PROGRAM SlowPRG_1
VAR
	bolPlcStartupDone: BOOL := FALSE;
	bolHostInitDone : BOOL := FALSE;
	bolInitDone : BOOL := FALSE;
	jj:INT;
	bolCtrlRst: BOOL;
	
	fbAlm_Man: FB_Alm_Man; // alarm manager
END_VAR

(*__________________________________________________________________________________________________
¦	
¦	Vistaprint Schweiz GmbH
¦	CH - 8401 Winterthur
¦
¦	www.vistaprint.ch - info@vistaprint.ch
¦___________________________________________________________________________________________________

Function desription:
call of all controller (FUB) for the slow task class.


History:
Version		Date			Author		Comment
---------------------------------------------------------------------------------------------------
0.00.1		24.05.2013		AVME/KVO	Start history
0.00.2		07.11.2013		AVME/KVO	Add local variabel fbAlm_Man, Add set all initialized controller FB the property of the alarm manager adress 
0.00.3		08.11.2013		AVME/KVO	global g_p_fbAlm_Man adress assigned
___________________________________________________________________________________________________*)


// -----------------------------------------------------------------------------------------------
// Initialize the PLC Parameter and check the PLC health
// -----------------------------------------------------------------------------------------------
IF (NOT bolPlcStartupDone) THEN

	// set all initialized controller FB the property of the alarm manager adress 
	Base_PLC.setAllCtrlAlarmFB(pCtrlInst := ADR(g_a_pCtrlInst[0]), pAlarmCtrl := ADR(fbAlm_Man), uinCtrlInstLength := INT_TO_UINT(E_CtrlId.E_CtrlIdMax));
	g_p_fbAlm_Man := ADR(fbAlm_Man);
	bolPlcStartupDone := TRUE;	
END_IF
// -----------------------------------------------------------------------------------------------


// -----------------------------------------------------------------------------------------------
// The host system is downloading all parameter at startup. 
// bolPlcStartupDone will be set to true after the Host is done with the initialization
// -----------------------------------------------------------------------------------------------
IF (bolPlcStartupDone AND (NOT bolHostInitDone) AND NOT bolInitDone) THEN
	bolHostInitDone := TRUE;
END_IF
// -----------------------------------------------------------------------------------------------


// -----------------------------------------------------------------------------------------------
// Start PLC code initialization
// -----------------------------------------------------------------------------------------------
IF NOT bolInitDone AND bolPlcStartupDone AND bolHostInitDone THEN
	
	// init	
	bolInitDone := TRUE;
END_IF
// -----------------------------------------------------------------------------------------------

// -----------------------------------------------------------------------------------------------
// Normal Run mode after all the initialization is done
// -----------------------------------------------------------------------------------------------
IF (bolInitDone AND bolPlcStartupDone AND bolHostInitDone) THEN
	
	//****************************************************************************************************
	// cyclic controller calls
	//****************************************************************************************************
	// call alarm message handler
	fbAlm_Man(bolCtrlRst:= bolCtrlRst);
	IF (bolCtrlRst) THEN
		FOR jj:=0 TO E_CtrlId.E_CtrlIdMax BY 1 DO
			IF (g_a_pCtrlCIf[jj]<>0) THEN // check if entry exist
				g_a_pCtrlCIf[jj]^.Job.bolAlmReset := TRUE;
			END_IF
		END_FOR
		bolCtrlRst := FALSE;
	END_IF

END_IF
// -----------------------------------------------------------------------------------------------

END_PROGRAM

(* stored: Version 1.1.0.1, ProductVersion 3.1.0.19
   POU SlowPRG_1: Id {f627bb3d-dce4-4692-ab49-07a63d91fd84} *)
